// TwinCAT 3 PLC project
// project tree:
//   POUs/ makeTupleStruct_1.TcPOU (not stored), proj0_TupleStruct_1.TcPOU, proj1_TupleStruct_1.TcPOU (not stored), makeTupleStruct_2.TcPOU, proj0_TupleStruct_2.TcPOU, proj1_TupleStruct_2.TcPOU, MAIN.TcPOU, makeArray0.TcPOU, makeArray1.TcPOU, normProjIdx.TcPOU (not stored), projArray1.TcPOU
//   DUTs/ STATE.TcDUT, enum_E.TcDUT, TupleStruct_1.TcDUT, TupleStruct_2.TcDUT
//   GVLs/ INPUTS.TcGVL (not stored), TIMERS.TcGVL (not stored)

// ---- DUTs/STATE.TcDUT

      TYPE STATE:
    STRUCT
        curTime: LREAL;
        dvar_M_aut_tii AT %Q*: TupleStruct_1;
        dvar_M_aut_ltii AT %Q*: ARRAY[0..1] of TupleStruct_1;
        dvar_M_aut_tlili AT %Q*: TupleStruct_2;
        dvar_M_aut_i AT %Q*: DINT;
        dvar_M_aut_j AT %Q*: DINT;
        dvar_M_aut AT %Q*: enum_E;
    END_STRUCT
END_TYPE

// ---- DUTs/enum_E.TcDUT
TYPE enum_E:
    (elit_l1, elit_l2, elit_l3, elit_l4, elit_l5);
END_TYPE

// ---- DUTs/TupleStruct_1.TcDUT

      TYPE TupleStruct_1:
    STRUCT
        field0: DINT;
        field1: DINT;
    END_STRUCT
END_TYPE

// ---- DUTs/TupleStruct_2.TcDUT

      TYPE TupleStruct_2:
    STRUCT
        field0: ARRAY[0..1] of DINT;
        field1: ARRAY[0..1] of DINT;
    END_STRUCT
END_TYPE

// ---- POUs/proj0_TupleStruct_1.TcPOU

      FUNCTION proj0_TupleStruct_1: DINT
VAR_INPUT
    tuple: TupleStruct_1;
END_VAR


        proj0_TupleStruct_1 := tuple.field0;

END_FUNCTION

// ---- POUs/makeTupleStruct_2.TcPOU
FUNCTION makeTupleStruct_2: TupleStruct_2
VAR_INPUT
    field0: ARRAY[0..1] of DINT;
    field1: ARRAY[0..1] of DINT;
END_VAR
VAR
    rslt: TupleStruct_2;
END_VAR

rslt.field0 := field0;
rslt.field1 := field1;
makeTupleStruct_2 := rslt;

END_FUNCTION

// ---- POUs/proj0_TupleStruct_2.TcPOU
FUNCTION proj0_TupleStruct_2: ARRAY[0..1] of DINT
VAR_INPUT
    tuple: TupleStruct_2;
END_VAR

proj0_TupleStruct_2 := tuple.field0;

END_FUNCTION

// ---- POUs/proj1_TupleStruct_2.TcPOU
FUNCTION proj1_TupleStruct_2: ARRAY[0..1] of DINT
VAR_INPUT
    tuple: TupleStruct_2;
END_VAR

proj1_TupleStruct_2 := tuple.field1;

END_FUNCTION

// ---- POUs/MAIN.TcPOU

      PROGRAM MAIN
VAR_OUTPUT
    timerValue0: TIME;
    timerValue1: TIME;
END_VAR
VAR
    cnt: LINT;
    first: BOOL := TRUE;
    curTimerValue: TIME;
    state0: STATE;
    curTime: LREAL;
    loopsKilled: LINT;
END_VAR
VAR_TEMP
    lastTimerValue: TIME;
    curDeltaTime: TIME;
    curDeltaSecs: LREAL;
    state1: STATE;
    progress: BOOL;
    loopCount: INT;
END_VAR


        
// Handle 'time' and cycle time.
cnt := cnt + 1;

timer0(IN := curTimer = 0, PT := T#1D);
timer1(IN := curTimer = 1, PT := T#1D);
timerValue0 := timer0.ET;
timerValue1 := timer1.ET;

lastTimerValue := curTimerValue;
IF curTimer = 0 THEN
    curTimerValue := timerValue0;
ELSE
    curTimerValue := timerValue1;
END_IF;
curDeltaTime := curTimerValue - lastTimerValue;
curDeltaSecs := TIME_TO_LREAL(curDeltaTime) / 1000;
curTime := curTime + curDeltaSecs;

IF cnt MOD 10 = 0 THEN
    curTimer := 1 - curTimer;
    curTimerValue := T#0S;
    timer0(IN := curTimer = 0, PT := T#1D);
    timer1(IN := curTimer = 1, PT := T#1D);
    timerValue0 := timer0.ET;
    timerValue1 := timer1.ET;
END_IF;

IF first THEN
    first := FALSE;

    // Initialize state variables for initial state.
    state0.dvar_M_aut_tii := makeTupleStruct_1(1, 2);
    state0.dvar_M_aut_ltii := makeArray0(makeTupleStruct_1(3, 4), makeTupleStruct_1(5, 6));
    state0.dvar_M_aut_tlili := makeTupleStruct_2(makeArray1(7, 8), makeArray1(9, 10));
    state0.dvar_M_aut_i := 11;
    state0.dvar_M_aut_j := 12;
    state0.dvar_M_aut := elit_l1;
ELSE
    // Update continuous variables for time delay.

    state0.curTime := curTime;
END_IF;

// Event loop.
WHILE TRUE DO
    progress := FALSE;

    // Event "tau".
    IF NOT progress THEN
        IF (state0.dvar_M_aut) = (elit_l1) THEN
            progress := TRUE;
            state1 := state0;

            state1.dvar_M_aut_i := proj1_TupleStruct_1(state0.dvar_M_aut_ltii[normProjIdx(0, 2)]);
            state1.dvar_M_aut_j := projArray1(proj1_TupleStruct_2(state0.dvar_M_aut_tlili), -1);
            state1.dvar_M_aut := elit_l2;

            state0 := state1;
        END_IF;
    END_IF;

    // Event "tau".
    IF NOT progress THEN
        IF (state0.dvar_M_aut) = (elit_l2) THEN
            progress := TRUE;
            state1 := state0;

            state1.dvar_M_aut_ltii[normProjIdx(-1, 2)].field0 := 13;
            state1.dvar_M_aut_tlili.field0[normProjIdx(-1, 2)] := 14;
            state1.dvar_M_aut := elit_l3;

            state0 := state1;
        END_IF;
    END_IF;

    // Event "tau".
    IF NOT progress THEN
        IF (state0.dvar_M_aut) = (elit_l3) THEN
            progress := TRUE;
            state1 := state0;

            state1.dvar_M_aut_ltii[normProjIdx(0, 2)] := state0.dvar_M_aut_tii;
            state1.dvar_M_aut := elit_l4;

            state0 := state1;
        END_IF;
    END_IF;

    // Event "tau".
    IF NOT progress THEN
        IF (state0.dvar_M_aut) = (elit_l4) THEN
            progress := TRUE;
            state1 := state0;

            state1.dvar_M_aut_tii := state0.dvar_M_aut_ltii[normProjIdx(1, 2)];
            state1.dvar_M_aut := elit_l5;

            state0 := state1;
        END_IF;
    END_IF;

    // Done with events?
    IF NOT progress THEN
        EXIT;
    END_IF;

    // Protect against events that are always enabled.
    loopCount := loopCount + 1;
    IF loopCount >= 100 THEN
        loopsKilled := loopsKilled + 1;
        EXIT;
    END_IF;
END_WHILE;

END_PROGRAM

// ---- POUs/makeArray0.TcPOU
FUNCTION makeArray0: ARRAY[0..1] of TupleStruct_1
VAR_INPUT
    elem0: TupleStruct_1;
    elem1: TupleStruct_1;
END_VAR
VAR
    rslt: ARRAY[0..1] of TupleStruct_1;
END_VAR

rslt[0] := elem0;
rslt[1] := elem1;
makeArray0 := rslt;

END_FUNCTION

// ---- POUs/makeArray1.TcPOU
FUNCTION makeArray1: ARRAY[0..1] of DINT
VAR_INPUT
    elem0: DINT;
    elem1: DINT;
END_VAR
VAR
    rslt: ARRAY[0..1] of DINT;
END_VAR

rslt[0] := elem0;
rslt[1] := elem1;
makeArray1 := rslt;

END_FUNCTION

// ---- POUs/projArray1.TcPOU

      FUNCTION projArray1: DINT
VAR_INPUT
    arr: ARRAY[0..1] of DINT;
    idx: DINT;
END_VAR


        projArray1 := arr[normProjIdx(idx, 2)];

END_FUNCTION
